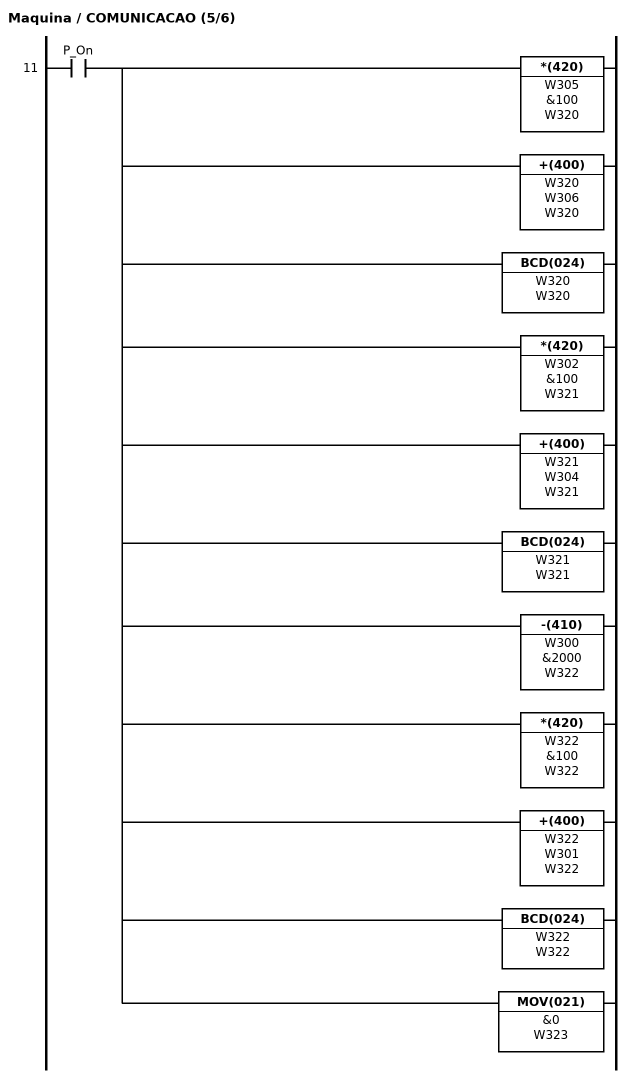
; [picture p24: Maquina / COMUNICACAO, rungs 11-11]
; rung 11
LD P_On
*(420) W305 &100 W320
+(400) W320 W306 W320
BCD(024) W320 W320
*(420) W302 &100 W321
+(400) W321 W304 W321
BCD(024) W321 W321
-(410) W300 &2000 W322
*(420) W322 &100 W322
+(400) W322 W301 W322
BCD(024) W322 W322
MOV(021) &0 W323

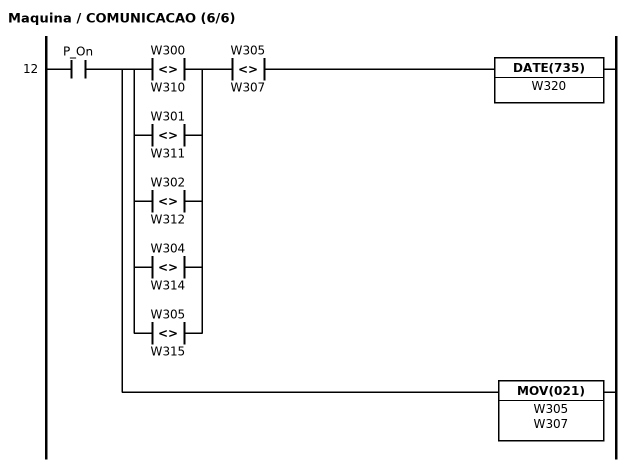
; rung 12
LD P_On
OUT TR0
LD<>(305) W300 W310
OR<>(305) W301 W311
OR<>(305) W302 W312
OR<>(305) W304 W314
OR<>(305) W305 W315
ANDLD
AND<>(305) W305 W307
DATE(735) W320
LD TR0
MOV(021) W305 W307

### Section TASK_CONTROL

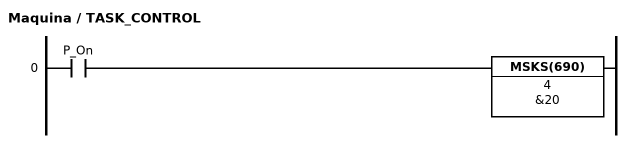
; rung 0
LD P_On
MSKS(690) 4 &20

### Section END
; rung 0
END(001)

## Program Inicializa_strings (cyclic task 127)
Local symbols
ano H130 STRING[2]
data_hora A351 WORD[3]
dia H126 STRING[2]
hora H124 STRING[2]
m_dlog_event_file_name W125 STRING[8]  ; Nome do ficheiro de datalogger
m_dlog_hum_file_name W135 STRING[8]  ; Nome do ficheiro de datalogger
m_dlog_maq_file_name W120 STRING[8]  ; Nome do ficheiro de datalogger
m_dlog_maq_name W110 STRING[10]  ; Nome da maquina
m_dlog_temp_file_name W130 STRING[8]  ; Nome do ficheiro de datalogger
mes H128 STRING[2]
minutos H122 STRING[2]
segundos H120 STRING[2]
str_data_hora H100 STRING[30]  ; String data/hora para datalogger
(*DATA/HORA PARA DATALOGGER*)
IF P_0_1ms=TRUE THEN
	minutos:=left (word_to_string(data_hora[0]),2);
	segundos:=right (word_to_string(data_hora[0]),2);
	dia:=left (word_to_string(data_hora[1]),2);
	hora:=right (word_to_string(data_hora[1]),2);
	ano:=left (word_to_string(data_hora[2]),2);
	mes:=right (word_to_string(data_hora[2]),2);
ELSE
	str_data_hora:= '20'+ano+'-'+mes+'-'+dia+' '+hora+':'+minutos+':'+segundos;
END_IF;

(*NOMES DOS FICHEIROS*)
(*************************************************************************************)

m_dlog_maq_name:= '6';	

m_dlog_maq_file_name:= '\PROG_6';	
m_dlog_event_file_name:= '\EVEN_6';
m_dlog_temp_file_name:= '\TEMP_6';
m_dlog_hum_file_name:= '\HUMI_6';

## Program CAUDAIS (interrupt task 2)
Local symbols
ft01 D700 STRUCT s_caudal  ; Caudalímetro
ft02 D720 STRUCT s_caudal  ; Caudalímetro
ft03 D740 STRUCT s_caudal  ; Caudalímetro
ft04 D760 STRUCT s_caudal  ; Caudalímetro
ft05 D780 STRUCT s_caudal  ; Caudalímetro
om5_injecta 2.15 BOOL  ; Pistola 5
tti1 1.00 BOOL  ; Caudalimetro 1
tti2 1.01 BOOL  ; Caudalimetro 2
tti3 1.02 BOOL  ; Caudalimetro 3
tti4 1.03 BOOL  ; Caudalimetro 4
tti5 1.04 BOOL  ; Caudalimetro 5

### Section M_CAUDAL

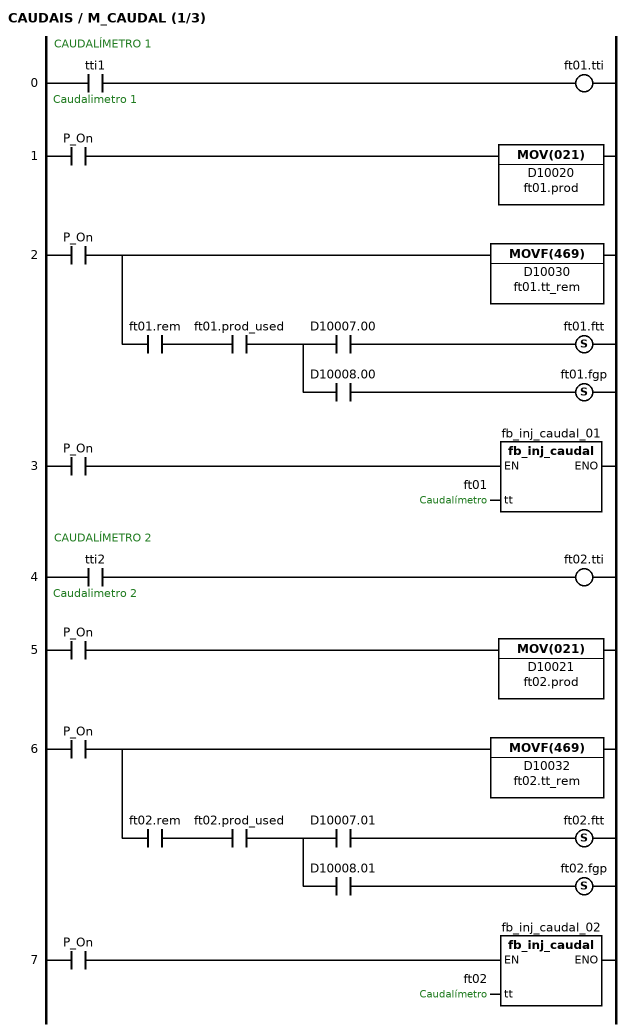
; rung 0: CAUDALÍMETRO 1
!LD tti1  ; Caudalimetro 1
OUT ft01.tti
; rung 1
LD P_On
MOV(021) D10020 ft01.prod
; rung 2
LD P_On
MOVF(469) D10030 ft01.tt_rem
AND ft01.rem
AND ft01.prod_used
OUT TR0
AND D10007.00
SET ft01.ftt
LD TR0
AND D10008.00
SET ft01.fgp
; rung 3
LD P_On
CALL fb_inj_caudal_01 : fb_inj_caudal (tt := ft01)  ; Caudalímetro
; rung 4: CAUDALÍMETRO 2
!LD tti2  ; Caudalimetro 2
OUT ft02.tti
; rung 5
LD P_On
MOV(021) D10021 ft02.prod
; rung 6
LD P_On
MOVF(469) D10032 ft02.tt_rem
AND ft02.rem
AND ft02.prod_used
OUT TR0
AND D10007.01
SET ft02.ftt
LD TR0
AND D10008.01
SET ft02.fgp
; rung 7
LD P_On
CALL fb_inj_caudal_02 : fb_inj_caudal (tt := ft02)  ; Caudalímetro

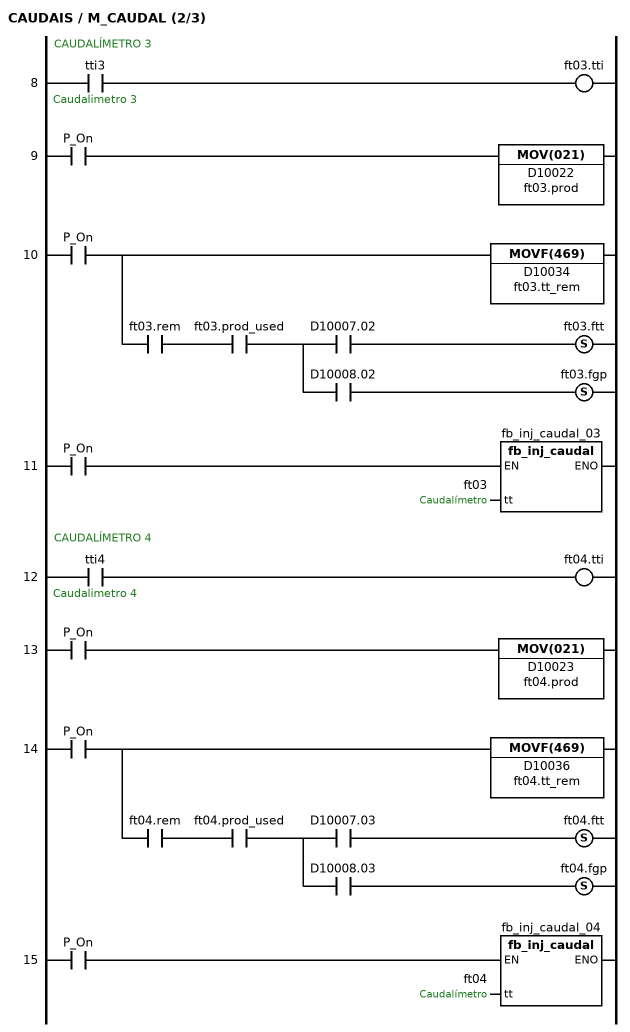
; rung 8: CAUDALÍMETRO 3
!LD tti3  ; Caudalimetro 3
OUT ft03.tti
; rung 9
LD P_On
MOV(021) D10022 ft03.prod
; rung 10
LD P_On
MOVF(469) D10034 ft03.tt_rem
AND ft03.rem
AND ft03.prod_used
OUT TR0
AND D10007.02
SET ft03.ftt
LD TR0
AND D10008.02
SET ft03.fgp
; rung 11
LD P_On
CALL fb_inj_caudal_03 : fb_inj_caudal (tt := ft03)  ; Caudalímetro
; rung 12: CAUDALÍMETRO 4
!LD tti4  ; Caudalimetro 4
OUT ft04.tti
; rung 13
LD P_On
MOV(021) D10023 ft04.prod
; rung 14
LD P_On
MOVF(469) D10036 ft04.tt_rem
AND ft04.rem
AND ft04.prod_used
OUT TR0
AND D10007.03
SET ft04.ftt
LD TR0
AND D10008.03
SET ft04.fgp
; rung 15
LD P_On
CALL fb_inj_caudal_04 : fb_inj_caudal (tt := ft04)  ; Caudalímetro

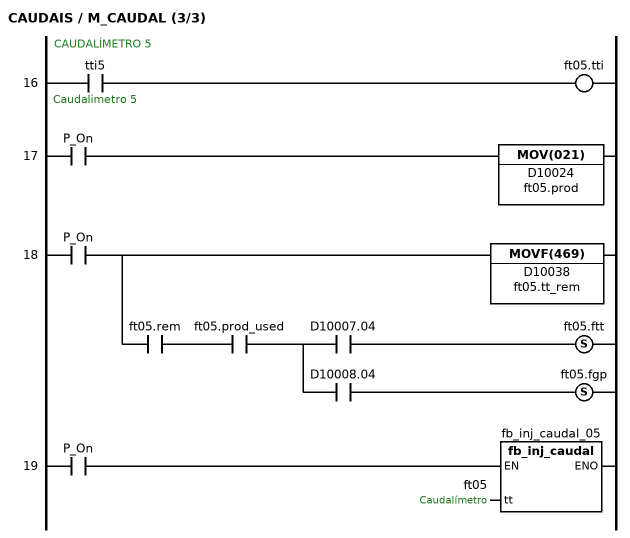
; rung 16: CAUDALÍMETRO 5
!LD tti5  ; Caudalimetro 5
OUT ft05.tti
; rung 17
LD P_On
MOV(021) D10024 ft05.prod
; rung 18
LD P_On
MOVF(469) D10038 ft05.tt_rem
AND ft05.rem
AND ft05.prod_used
OUT TR0
AND D10007.04
SET ft05.ftt
LD TR0
AND D10008.04
SET ft05.fgp
; rung 19
LD P_On
CALL fb_inj_caudal_05 : fb_inj_caudal (tt := ft05)  ; Caudalímetro

### Section END
; rung 0
END(001)

## Function block ExeTimeCalc
VAR_INPUT
  Enable : BOOL;
END_VAR
VAR_OUTPUT
  TotalTime : INT;
  CDT : INT;
END_VAR
VAR_IN_OUT
  prg : s_of_prg;
END_VAR
VAR
  itr : INT;
  ElapsedTime : INT;
  Stp : ARRAY[0..11] OF s_of_pss;
END_VAR
TotalTime:= 0;
ElapsedTime:= 0;

Stp[0].p1:= prg.pss[0].p1; Stp[0].tt:= prg.pss[0].tt; Stp[0].uni:= prg.pss[0].uni;
Stp[1].p1:= prg.pss[1].p1; Stp[1].tt:= prg.pss[1].tt; Stp[1].uni:= prg.pss[1].uni;
Stp[2].p1:= prg.pss[2].p1; Stp[2].tt:= prg.pss[2].tt;Stp[2].uni:= prg.pss[2].uni;
Stp[3].p1:= prg.pss[3].p1; Stp[3].tt:= prg.pss[3].tt; Stp[3].uni:= prg.pss[3].uni;
Stp[4].p1:= prg.pss[4].p1; Stp[4].tt:= prg.pss[4].tt; Stp[4].uni:= prg.pss[4].uni;
Stp[5].p1:= prg.pss[5].p1; Stp[5].tt:= prg.pss[5].tt; Stp[5].uni:= prg.pss[5].uni;
Stp[6].p1:= prg.pss[6].p1; Stp[6].tt:= prg.pss[6].tt; Stp[6].uni:= prg.pss[6].uni;
Stp[7].p1:= prg.pss[7].p1; Stp[7].tt:= prg.pss[7].tt; Stp[7].uni:= prg.pss[7].uni;
Stp[8].p1:= prg.pss[8].p1; Stp[8].tt:= prg.pss[8].tt; Stp[8].uni:= prg.pss[8].uni;
Stp[9].p1:= prg.pss[9].p1; Stp[9].tt:= prg.pss[9].tt; Stp[9].uni:= prg.pss[9].uni;
Stp[10].p1:= prg.pss[10].p1; Stp[10].tt:= prg.pss[10].tt; Stp[10].uni:= prg.pss[10].uni;
Stp[11].p1:= prg.pss[11].p1; Stp[11].tt:= prg.pss[11].tt; Stp[11].uni:= prg.pss[11].uni;

IF Enable THEN
	FOR itr:=0 TO 11 DO
		IF Stp[ itr ].uni=12 THEN
			TotalTime:=TotalTime+ Stp[ itr ].p1;
			ElapsedTime:= ElapsedTime+REAL_TO_INT(Stp[ itr ].tt);
		END_IF;
	END_FOR;
END_IF;
	
CDT := TotalTime - ElapsedTime;

## Function block fb_CopySteps
VAR_INPUT
  Rcp_Ok : BOOL;
END_VAR
VAR_IN_OUT
  Recipe : s_of;
  Steps : ARRAY[0..11] OF s_Steps;
END_VAR
(*Programa*)
Recipe.prg.pss[0].f:=Steps[0].f;
Recipe.prg.pss[0].p1:=Steps[0].p1;
Recipe.prg.pss[0].p2:=Steps[0].p2;
Recipe.prg.pss[0].uni:=0;
Recipe.prg.pss[0].uni:=12;
CASE Recipe.prg.pss[0].f OF
	40:Recipe.prg.pss[0].uni:=9;
END_CASE;

Recipe.prg.pss[1].f:=Steps[1].f;
Recipe.prg.pss[1].p1:=Steps[1].p1;
Recipe.prg.pss[1].p2:=Steps[1].p2;
Recipe.prg.pss[1].uni:=0;
Recipe.prg.pss[1].uni:=12;
CASE Recipe.prg.pss[1].f OF
	40:Recipe.prg.pss[1].uni:=9;
END_CASE;

Recipe.prg.pss[2].f:=Steps[2].f;
Recipe.prg.pss[2].p1:=Steps[2].p1;
Recipe.prg.pss[2].p2:=Steps[2].p2;
Recipe.prg.pss[2].uni:=0;
Recipe.prg.pss[2].uni:=12;
CASE Recipe.prg.pss[2].f OF
	40:Recipe.prg.pss[2].uni:=9;
END_CASE;

Recipe.prg.pss[3].f:=Steps[3].f;
Recipe.prg.pss[3].p1:=Steps[3].p1;
Recipe.prg.pss[3].p2:=Steps[3].p2;
Recipe.prg.pss[3].uni:=0;
Recipe.prg.pss[3].uni:=12;
CASE Recipe.prg.pss[3].f OF
	40:Recipe.prg.pss[3].uni:=9;
END_CASE;

Recipe.prg.pss[4].f:=Steps[4].f;
Recipe.prg.pss[4].p1:=Steps[4].p1;
Recipe.prg.pss[4].p2:=Steps[4].p2;
Recipe.prg.pss[4].uni:=0;
Recipe.prg.pss[4].uni:=12;
CASE Recipe.prg.pss[4].f OF
	40:Recipe.prg.pss[4].uni:=9;
END_CASE;

Recipe.prg.pss[5].f:=Steps[5].f;
Recipe.prg.pss[5].p1:=Steps[5].p1;
Recipe.prg.pss[5].p2:=Steps[5].p2;
Recipe.prg.pss[5].uni:=0;
Recipe.prg.pss[5].uni:=12;
CASE Recipe.prg.pss[5].f OF
	40:Recipe.prg.pss[5].uni:=9;
END_CASE;

Recipe.prg.pss[6].f:=Steps[6].f;
Recipe.prg.pss[6].p1:=Steps[6].p1;
Recipe.prg.pss[6].p2:=Steps[6].p2;
Recipe.prg.pss[6].uni:=0;
Recipe.prg.pss[6].uni:=12;
CASE Recipe.prg.pss[6].f OF
	40:Recipe.prg.pss[6].uni:=9;
END_CASE;

Recipe.prg.pss[7].f:=Steps[7].f;
Recipe.prg.pss[7].p1:=Steps[7].p1;
Recipe.prg.pss[7].p2:=Steps[7].p2;
Recipe.prg.pss[7].uni:=0;
Recipe.prg.pss[7].uni:=12;
CASE Recipe.prg.pss[7].f OF
	40:Recipe.prg.pss[7].uni:=9;
END_CASE;

Recipe.prg.pss[8].f:=Steps[8].f;
Recipe.prg.pss[8].p1:=Steps[8].p1;
Recipe.prg.pss[8].p2:=Steps[8].p2;
Recipe.prg.pss[8].uni:=0;
Recipe.prg.pss[8].uni:=12;
CASE Recipe.prg.pss[8].f OF
	40:Recipe.prg.pss[8].uni:=9;
END_CASE;

Recipe.prg.pss[9].f:=Steps[9].f;
Recipe.prg.pss[9].p1:=Steps[9].p1;
Recipe.prg.pss[9].p2:=Steps[9].p2;
Recipe.prg.pss[9].uni:=0;
Recipe.prg.pss[9].uni:=12;
CASE Recipe.prg.pss[9].f OF
	40:Recipe.prg.pss[9].uni:=9;
END_CASE;

Recipe.prg.pss[10].f:=Steps[9].f;
Recipe.prg.pss[10].p1:=Steps[9].p1;
Recipe.prg.pss[10].p2:=Steps[9].p2;
Recipe.prg.pss[10].uni:=0;
Recipe.prg.pss[10].uni:=12;
CASE Recipe.prg.pss[10].f OF
	40:Recipe.prg.pss[10].uni:=9;
END_CASE;

Recipe.prg.pss[11].f:=Steps[9].f;
Recipe.prg.pss[11].p1:=Steps[9].p1;
Recipe.prg.pss[11].p2:=Steps[9].p2;
Recipe.prg.pss[11].uni:=0;
Recipe.prg.pss[11].uni:=12;
CASE Recipe.prg.pss[11].f OF
	40:Recipe.prg.pss[11].uni:=9;
END_CASE;

Recipe.dados:= Rcp_Ok;

## Function block fb_f_aquece
; FUNÇÃO AQUECIMENTO USANDO TC104 - Faz a função de aquecimento usando uma carta TC104 com PID
VAR_IN_OUT
  maq : s_maquina;  (* Dados da maquina *)
  aquece : s_f_aquece;  (* Dados da função de aquecimento *)
  aspira : s_f_aspira;  (* Dados da função de aspiração *)
END_VAR
VAR
  tm01 : TIMER;
  sp_hh : REAL;  (* Valor superior do setpoint *)
  sp_ll : REAL;  (* Valor inferior do setpoint *)
  p1 : REAL;  (* Parametro 1 da função em REAL *)
  sp_ft : UDINT;
  tm02 : TIMER;
  tm03 : TIMER;
  tm04 : TIMER;
  p1_end : REAL;  (* Valor apartir do qual deixa de aquecer. *)
END_VAR

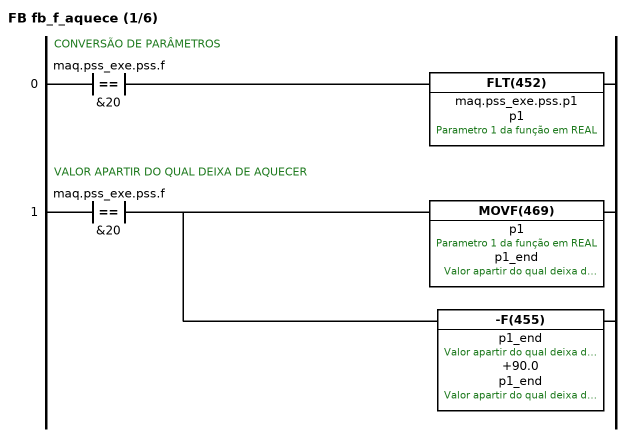
; rung 0: CONVERSÃO DE PARÂMETROS
LD=(300) maq.pss_exe.pss.f &20
FLT(452) maq.pss_exe.pss.p1 p1  ; Parametro 1 da função em REAL
; rung 1: VALOR APARTIR DO QUAL DEIXA DE AQUECER
LD=(300) maq.pss_exe.pss.f &20
MOVF(469) p1 p1_end  ; Parametro 1 da função em REAL, Valor apartir do qual deixa de aquecer.
-F(455) p1_end +90.0 p1_end  ; Valor apartir do qual deixa de aquecer.

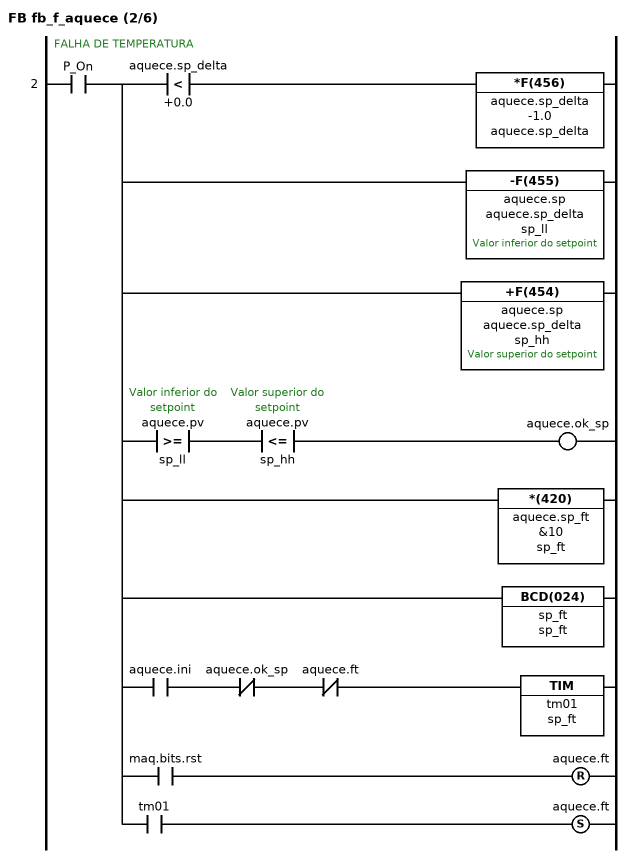
; rung 2: FALHA DE TEMPERATURA
LD P_On
OUT TR0
AND<F(331) aquece.sp_delta +0.0
*F(456) aquece.sp_delta -1.0 aquece.sp_delta
LD TR0
-F(455) aquece.sp aquece.sp_delta sp_ll  ; Valor inferior do setpoint
+F(454) aquece.sp aquece.sp_delta sp_hh  ; Valor superior do setpoint
AND>=F(334) aquece.pv sp_ll  ; Valor inferior do setpoint
AND<=F(332) aquece.pv sp_hh  ; Valor superior do setpoint
OUT aquece.ok_sp
LD TR0
*(420) aquece.sp_ft &10 sp_ft
BCD(024) sp_ft sp_ft
AND aquece.ini
ANDNOT aquece.ok_sp
ANDNOT aquece.ft
TIM tm01 sp_ft
LD TR0
AND maq.bits.rst
RSET aquece.ft
LD TR0
AND tm01
SET aquece.ft

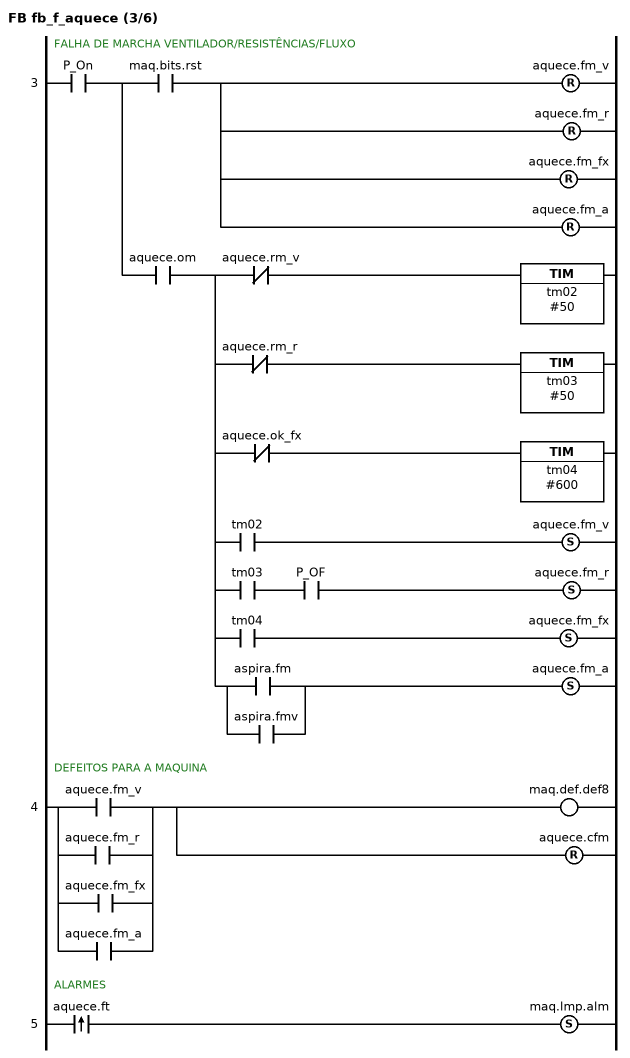
; rung 3: FALHA DE MARCHA VENTILADOR/RESISTÊNCIAS/FLUXO
LD P_On
OUT TR0
AND maq.bits.rst
RSET aquece.fm_v
RSET aquece.fm_r
RSET aquece.fm_fx
RSET aquece.fm_a
LD TR0
AND aquece.om
OUT TR1
ANDNOT aquece.rm_v
TIM tm02 #50
LD TR1
ANDNOT aquece.rm_r
TIM tm03 #50
LD TR1
ANDNOT aquece.ok_fx
TIM tm04 #600
LD TR1
AND tm02
SET aquece.fm_v
LD TR1
AND tm03
AND P_OF
SET aquece.fm_r
LD TR1
AND tm04
SET aquece.fm_fx
LD TR1
LD aspira.fm
OR aspira.fmv
ANDLD
SET aquece.fm_a
; rung 4: DEFEITOS PARA A MAQUINA
LD aquece.fm_v
OR aquece.fm_r
OR aquece.fm_fx
OR aquece.fm_a
OUT maq.def.def8
RSET aquece.cfm
; rung 5: ALARMES
@LD aquece.ft
SET maq.lmp.alm

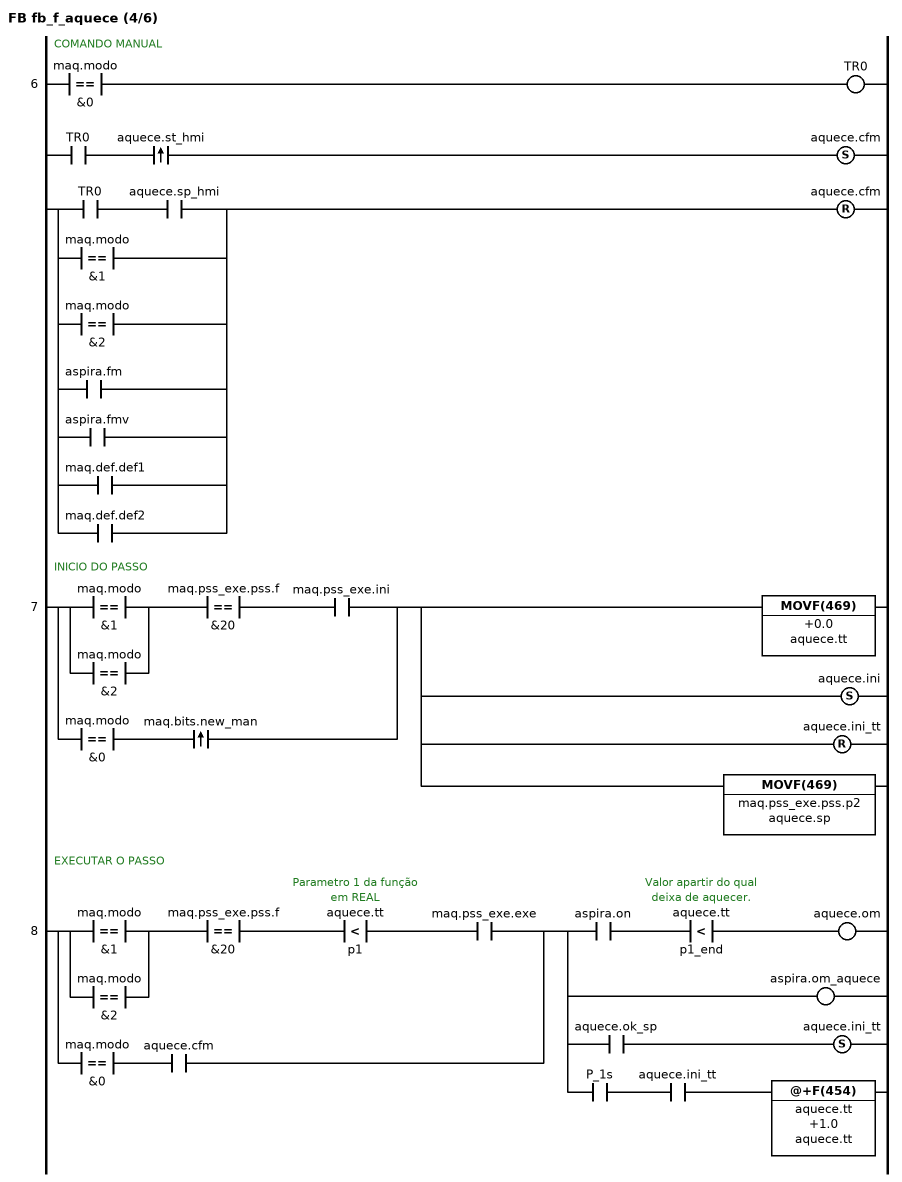
; rung 6: COMANDO MANUAL
LD=(300) maq.modo &0
OUT TR0
LD TR0
@AND aquece.st_hmi
SET aquece.cfm
LD TR0
AND aquece.sp_hmi
OR=(300) maq.modo &1
OR=(300) maq.modo &2
OR aspira.fm
OR aspira.fmv
OR maq.def.def1
OR maq.def.def2
RSET aquece.cfm
; rung 7: INICIO DO PASSO
LD=(300) maq.modo &1
OR=(300) maq.modo &2
AND=(300) maq.pss_exe.pss.f &20
AND maq.pss_exe.ini
LD=(300) maq.modo &0
@AND maq.bits.new_man
ORLD
MOVF(469) +0.0 aquece.tt
SET aquece.ini
RSET aquece.ini_tt
MOVF(469) maq.pss_exe.pss.p2 aquece.sp
; rung 8: EXECUTAR O PASSO
LD=(300) maq.modo &1
OR=(300) maq.modo &2
AND=(300) maq.pss_exe.pss.f &20
AND<F(331) aquece.tt p1  ; Parametro 1 da função em REAL
AND maq.pss_exe.exe
LD=(300) maq.modo &0
AND aquece.cfm
ORLD
OUT TR0
AND aspira.on
AND<F(331) aquece.tt p1_end  ; Valor apartir do qual deixa de aquecer.
OUT aquece.om
LD TR0
OUT aspira.om_aquece
AND aquece.ok_sp
SET aquece.ini_tt
LD TR0
AND P_1s
AND aquece.ini_tt
@+F(454) aquece.tt +1.0 aquece.tt

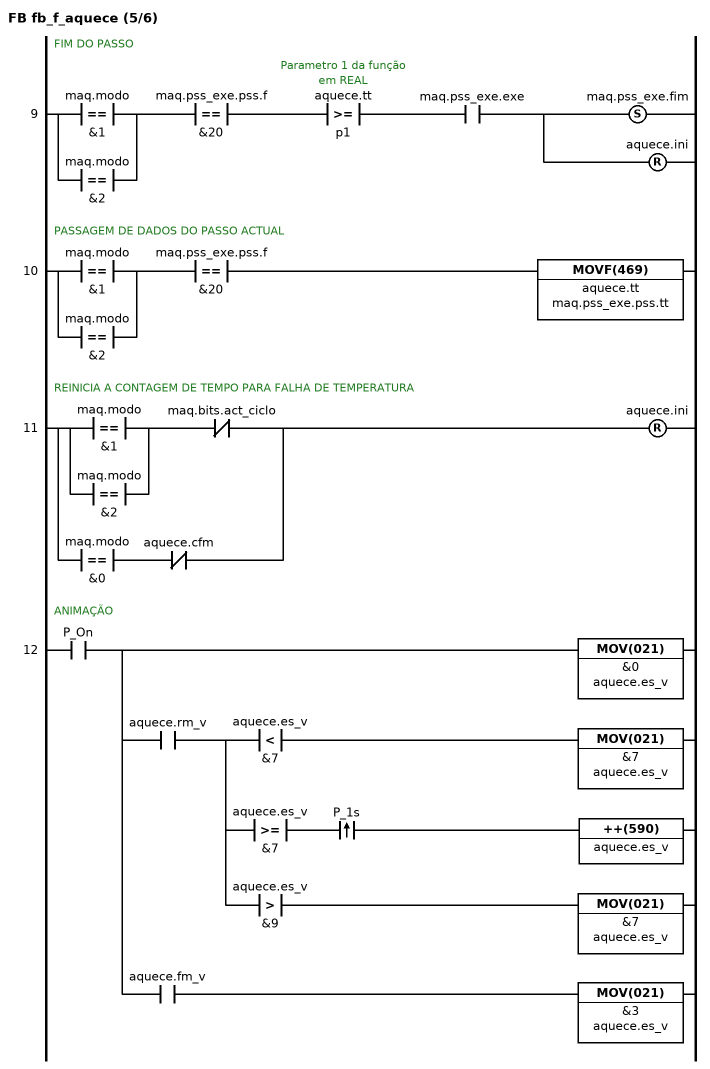
; rung 9: FIM DO PASSO
LD=(300) maq.modo &1
OR=(300) maq.modo &2
AND=(300) maq.pss_exe.pss.f &20
AND>=F(334) aquece.tt p1  ; Parametro 1 da função em REAL
AND maq.pss_exe.exe
SET maq.pss_exe.fim
RSET aquece.ini
; rung 10: PASSAGEM DE DADOS DO PASSO ACTUAL
LD=(300) maq.modo &1
OR=(300) maq.modo &2
AND=(300) maq.pss_exe.pss.f &20
MOVF(469) aquece.tt maq.pss_exe.pss.tt
; rung 11: REINICIA A CONTAGEM DE TEMPO PARA FALHA DE TEMPERATURA
LD=(300) maq.modo &1
OR=(300) maq.modo &2
ANDNOT maq.bits.act_ciclo
LD=(300) maq.modo &0
ANDNOT aquece.cfm
ORLD
RSET aquece.ini
; rung 12: ANIMAÇÃO
LD P_On
OUT TR0
MOV(021) &0 aquece.es_v
AND aquece.rm_v
OUT TR1
AND<(310) aquece.es_v &7
MOV(021) &7 aquece.es_v
LD TR1
AND>=(325) aquece.es_v &7
@AND P_1s
++(590) aquece.es_v
LD TR1
AND>(320) aquece.es_v &9
MOV(021) &7 aquece.es_v
LD TR0
AND aquece.fm_v
MOV(021) &3 aquece.es_v

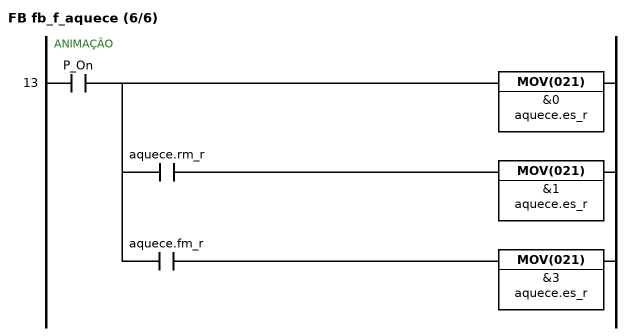
; rung 13: ANIMAÇÃO
LD P_On
OUT TR0
MOV(021) &0 aquece.es_r
AND aquece.rm_r
MOV(021) &1 aquece.es_r
LD TR0
AND aquece.fm_r
MOV(021) &3 aquece.es_r

## Function block fb_f_aspira
; FUNÇÃO ASPIRAÇÃO - Faz a função de aspiração. Controlo de inputs/outputs
VAR_IN_OUT
  maq : s_maquina;  (* Dados da maquina *)
  aspira : s_f_aspira;  (* Dados da função de aspiração *)
END_VAR
VAR
  tm01 : TIMER;
  tm02 : TIMER;
  p1 : REAL;  (* Parametro 1 da função em REAL *)
  tm03 : TIMER;
END_VAR

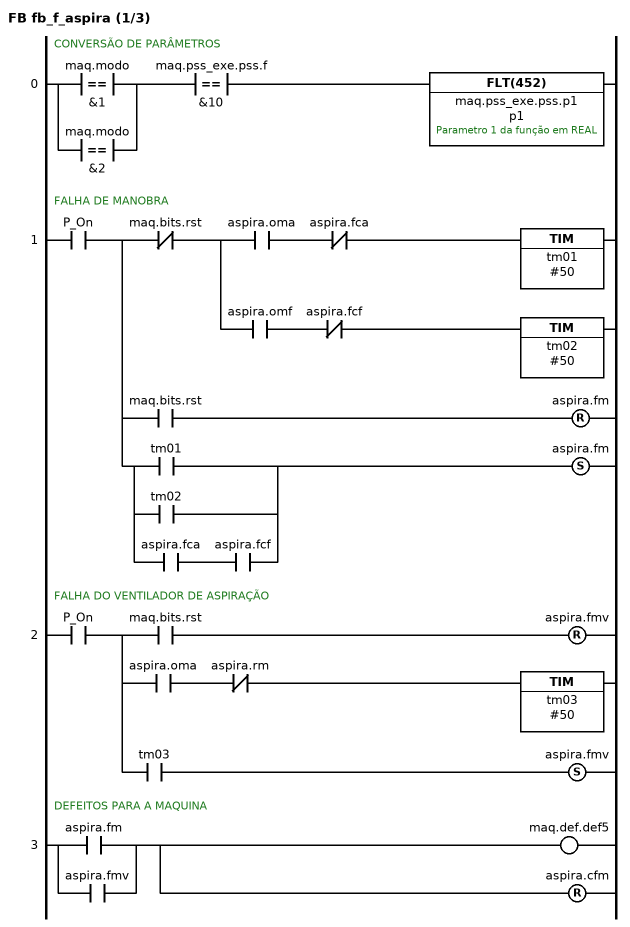
; rung 0: CONVERSÃO DE PARÂMETROS
LD=(300) maq.modo &1
OR=(300) maq.modo &2
AND=(300) maq.pss_exe.pss.f &10
FLT(452) maq.pss_exe.pss.p1 p1  ; Parametro 1 da função em REAL
; rung 1: FALHA DE MANOBRA
LD P_On
OUT TR0
ANDNOT maq.bits.rst
OUT TR1
AND aspira.oma
ANDNOT aspira.fca
TIM tm01 #50
LD TR1
AND aspira.omf
ANDNOT aspira.fcf
TIM tm02 #50
LD TR0
AND maq.bits.rst
RSET aspira.fm
LD TR0
LD tm01
OR tm02
LD aspira.fca
AND aspira.fcf
ORLD
ANDLD
SET aspira.fm
; rung 2: FALHA DO VENTILADOR DE ASPIRAÇÃO
LD P_On
OUT TR0
AND maq.bits.rst
RSET aspira.fmv
LD TR0
AND aspira.oma
ANDNOT aspira.rm
TIM tm03 #50
LD TR0
AND tm03
SET aspira.fmv
; rung 3: DEFEITOS PARA A MAQUINA
LD aspira.fm
OR aspira.fmv
OUT maq.def.def5
RSET aspira.cfm

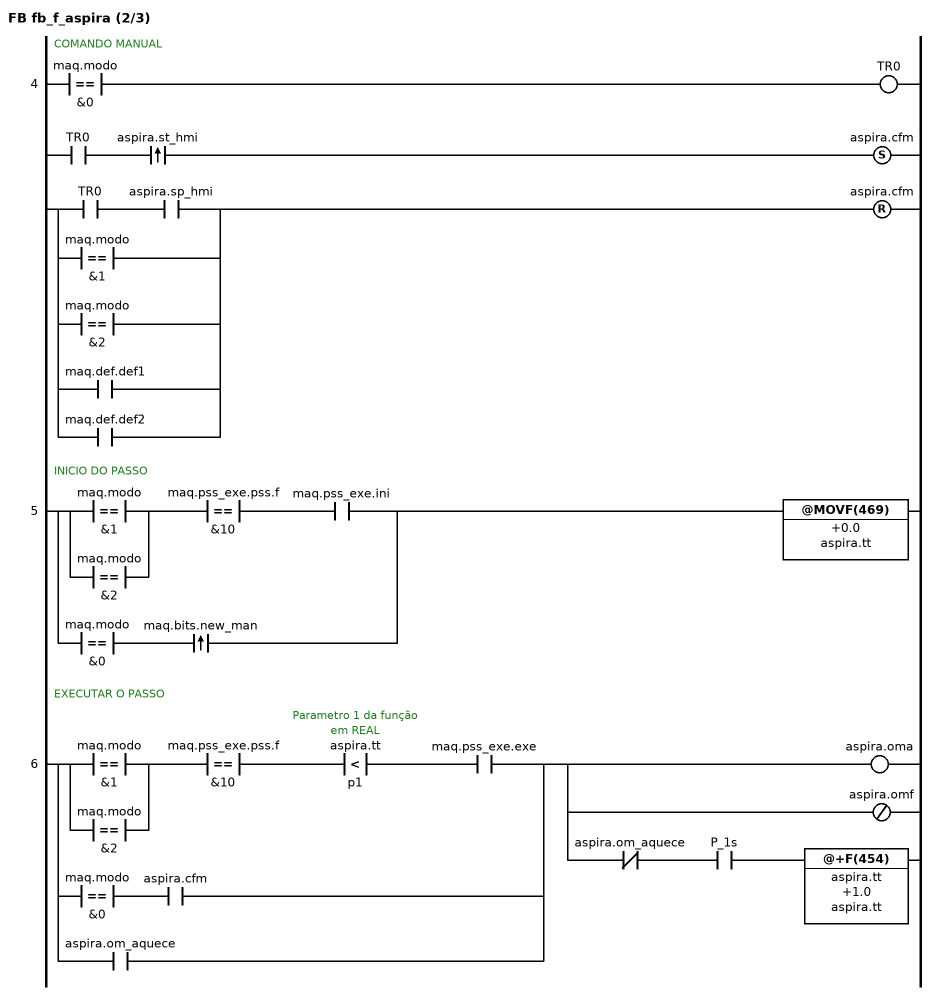
; rung 4: COMANDO MANUAL
LD=(300) maq.modo &0
OUT TR0
LD TR0
@AND aspira.st_hmi
SET aspira.cfm
LD TR0
AND aspira.sp_hmi
OR=(300) maq.modo &1
OR=(300) maq.modo &2
OR maq.def.def1
OR maq.def.def2
RSET aspira.cfm
; rung 5: INICIO DO PASSO
LD=(300) maq.modo &1
OR=(300) maq.modo &2
AND=(300) maq.pss_exe.pss.f &10
AND maq.pss_exe.ini
LD=(300) maq.modo &0
@AND maq.bits.new_man
ORLD
@MOVF(469) +0.0 aspira.tt
; rung 6: EXECUTAR O PASSO
LD=(300) maq.modo &1
OR=(300) maq.modo &2
AND=(300) maq.pss_exe.pss.f &10
AND<F(331) aspira.tt p1  ; Parametro 1 da função em REAL
AND maq.pss_exe.exe
LD=(300) maq.modo &0
AND aspira.cfm
ORLD
OR aspira.om_aquece
OUT aspira.oma
OUTNOT aspira.omf
ANDNOT aspira.om_aquece
AND P_1s
@+F(454) aspira.tt +1.0 aspira.tt

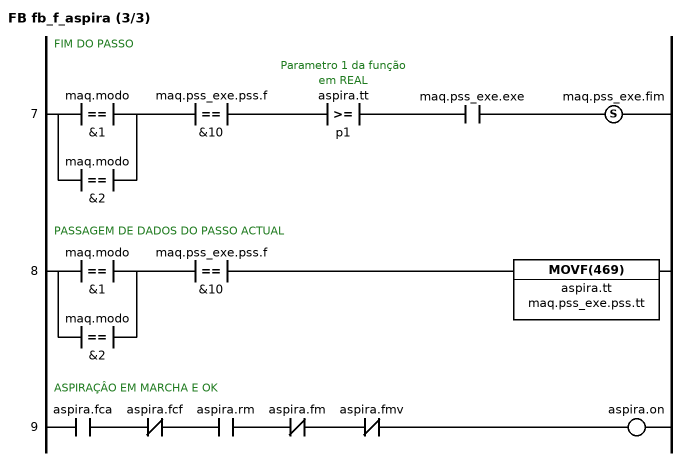
; rung 7: FIM DO PASSO
LD=(300) maq.modo &1
OR=(300) maq.modo &2
AND=(300) maq.pss_exe.pss.f &10
AND>=F(334) aspira.tt p1  ; Parametro 1 da função em REAL
AND maq.pss_exe.exe
SET maq.pss_exe.fim
; rung 8: PASSAGEM DE DADOS DO PASSO ACTUAL
LD=(300) maq.modo &1
OR=(300) maq.modo &2
AND=(300) maq.pss_exe.pss.f &10
MOVF(469) aspira.tt maq.pss_exe.pss.tt
; rung 9: ASPIRAÇÂO EM MARCHA E OK
LD aspira.fca
ANDNOT aspira.fcf
AND aspira.rm
ANDNOT aspira.fm
ANDNOT aspira.fmv
OUT aspira.on

## Function block fb_f_injecta
; FUNÇÃO INJECÇÃO - Faz a função de injecção
VAR_IN_OUT
  maq : s_maquina;  (* Dados da maquina *)
  injecta : s_f_injecta;  (* Dados da função de injecção *)
  caudal : s_caudal;  (* Dados do caudalímetro *)
END_VAR
VAR
  tm01 : TIMER;
END_VAR

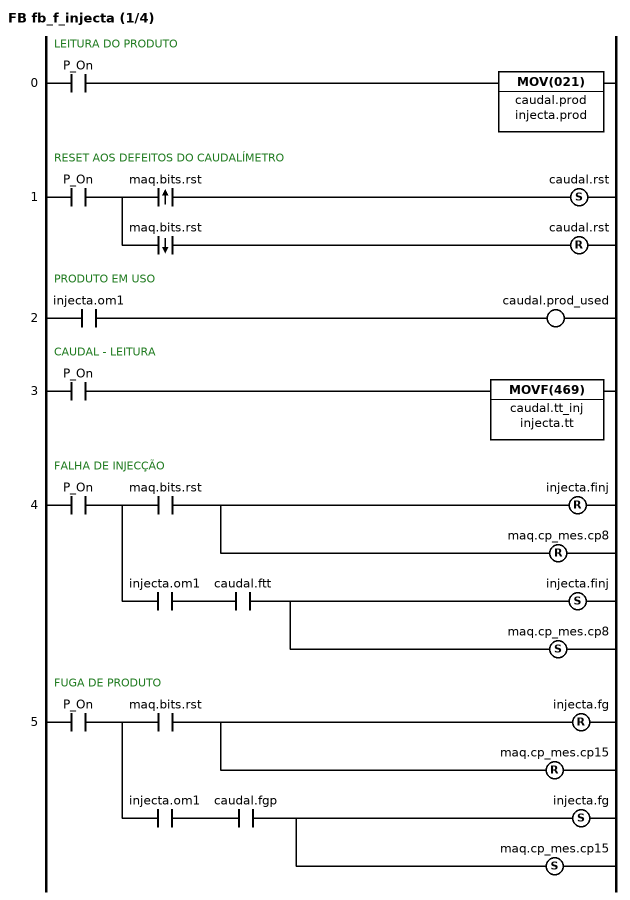
; rung 0: LEITURA DO PRODUTO
LD P_On
MOV(021) caudal.prod injecta.prod
; rung 1: RESET AOS DEFEITOS DO CAUDALÍMETRO
LD P_On
OUT TR0
@AND maq.bits.rst
SET caudal.rst
LD TR0
%AND maq.bits.rst
RSET caudal.rst
; rung 2: PRODUTO EM USO
LD injecta.om1
OUT caudal.prod_used
; rung 3: CAUDAL - LEITURA
LD P_On
MOVF(469) caudal.tt_inj injecta.tt
; rung 4: FALHA DE INJECÇÃO
LD P_On
OUT TR0
AND maq.bits.rst
RSET injecta.finj
RSET maq.cp_mes.cp8
LD TR0
AND injecta.om1
AND caudal.ftt
SET injecta.finj
SET maq.cp_mes.cp8
; rung 5: FUGA DE PRODUTO
LD P_On
OUT TR0
AND maq.bits.rst
RSET injecta.fg
RSET maq.cp_mes.cp15
LD TR0
AND injecta.om1
AND caudal.fgp
SET injecta.fg
SET maq.cp_mes.cp15

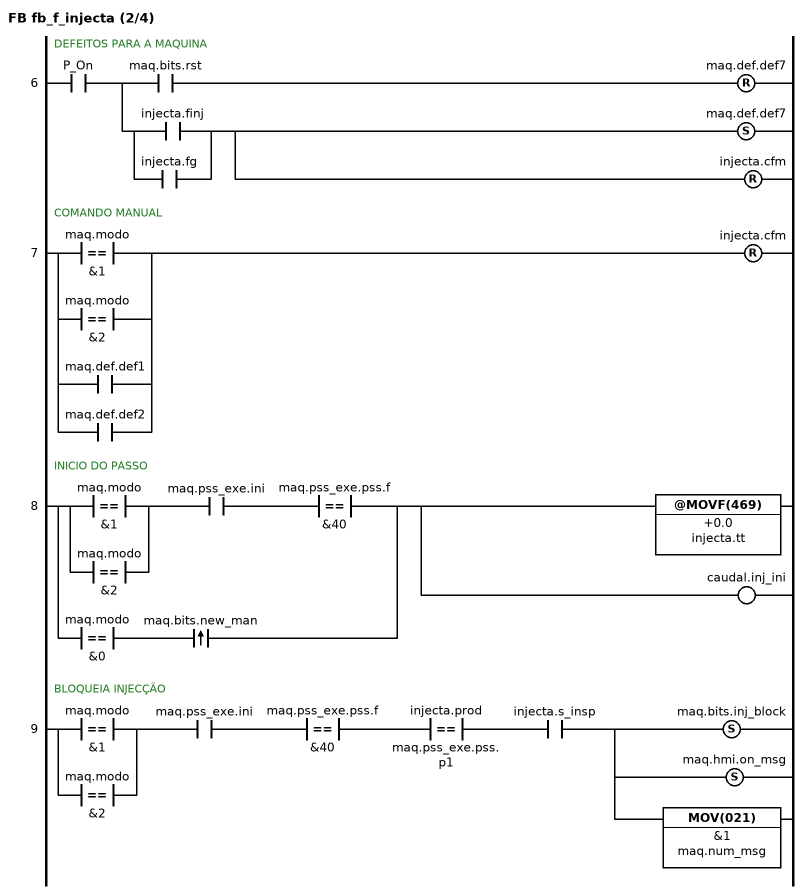
; rung 6: DEFEITOS PARA A MAQUINA
LD P_On
OUT TR0
AND maq.bits.rst
RSET maq.def.def7
LD TR0
LD injecta.finj
OR injecta.fg
ANDLD
SET maq.def.def7
RSET injecta.cfm
; rung 7: COMANDO MANUAL
LD=(300) maq.modo &1
OR=(300) maq.modo &2
OR maq.def.def1
OR maq.def.def2
RSET injecta.cfm
; rung 8: INICIO DO PASSO
LD=(300) maq.modo &1
OR=(300) maq.modo &2
AND maq.pss_exe.ini
AND=(300) maq.pss_exe.pss.f &40
LD=(300) maq.modo &0
@AND maq.bits.new_man
ORLD
@MOVF(469) +0.0 injecta.tt
OUT caudal.inj_ini
; rung 9: BLOQUEIA INJECÇÃO
LD=(300) maq.modo &1
OR=(300) maq.modo &2
AND maq.pss_exe.ini
AND=(300) maq.pss_exe.pss.f &40
AND=(300) injecta.prod maq.pss_exe.pss.p1
AND injecta.s_insp
SET maq.bits.inj_block
SET maq.hmi.on_msg
MOV(021) &1 maq.num_msg

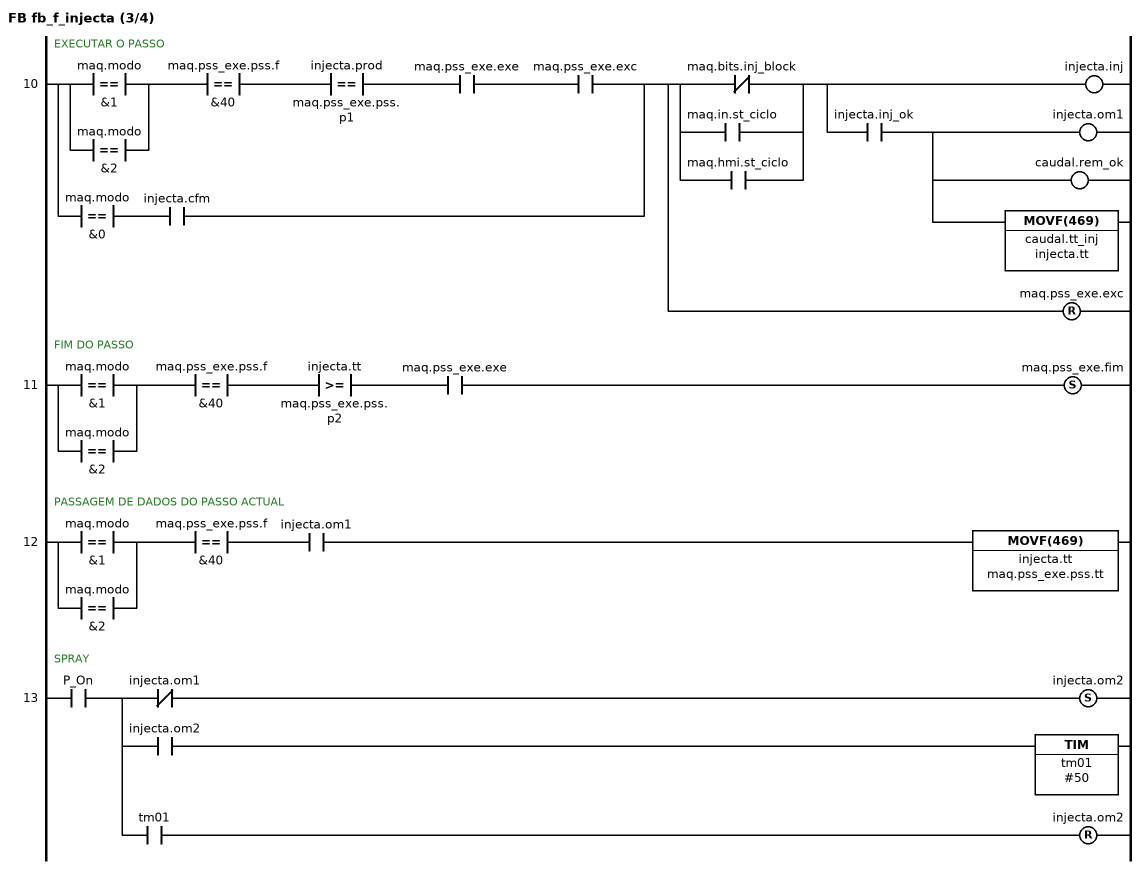
; rung 10: EXECUTAR O PASSO
LD=(300) maq.modo &1
OR=(300) maq.modo &2
AND=(300) maq.pss_exe.pss.f &40
AND=(300) injecta.prod maq.pss_exe.pss.p1
AND maq.pss_exe.exe
AND maq.pss_exe.exc
LD=(300) maq.modo &0
AND injecta.cfm
ORLD
OUT TR0
LDNOT maq.bits.inj_block
OR maq.in.st_ciclo
OR maq.hmi.st_ciclo
ANDLD
OUT injecta.inj
AND injecta.inj_ok
OUT injecta.om1
OUT caudal.rem_ok
MOVF(469) caudal.tt_inj injecta.tt
LD TR0
RSET maq.pss_exe.exc
; rung 11: FIM DO PASSO
LD=(300) maq.modo &1
OR=(300) maq.modo &2
AND=(300) maq.pss_exe.pss.f &40
AND>=F(334) injecta.tt maq.pss_exe.pss.p2
AND maq.pss_exe.exe
SET maq.pss_exe.fim
; rung 12: PASSAGEM DE DADOS DO PASSO ACTUAL
LD=(300) maq.modo &1
OR=(300) maq.modo &2
AND=(300) maq.pss_exe.pss.f &40
AND injecta.om1
MOVF(469) injecta.tt maq.pss_exe.pss.tt
; rung 13: SPRAY
LD P_On
OUT TR0
ANDNOT injecta.om1
SET injecta.om2
LD TR0
AND injecta.om2
TIM tm01 #50
LD TR0
AND tm01
RSET injecta.om2

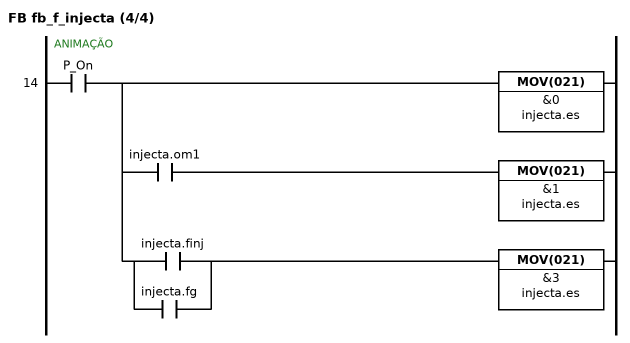
; rung 14: ANIMAÇÃO
LD P_On
OUT TR0
MOV(021) &0 injecta.es
AND injecta.om1
MOV(021) &1 injecta.es
LD TR0
LD injecta.finj
OR injecta.fg
ANDLD
MOV(021) &3 injecta.es

## Function block fb_f_injecta_man
; FUNÇÃO INJECÇÃO MANUAL - Faz a função de injecção manual (chamar após injecção auto)
VAR_IN_OUT
  maq : s_maquina;  (* Dados da maquina *)
END_VAR

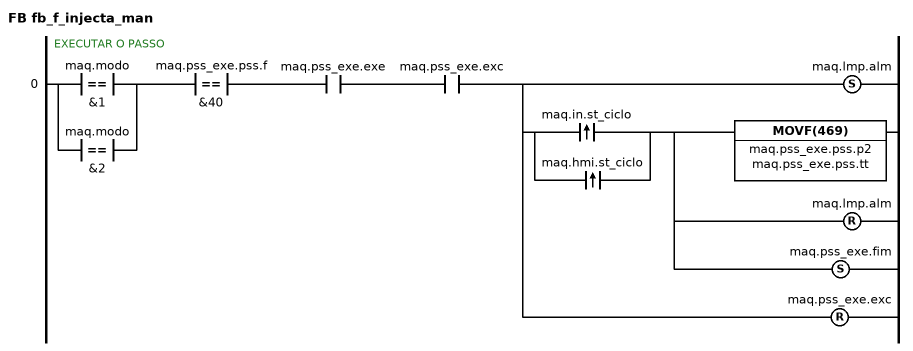
; rung 0: EXECUTAR O PASSO
LD=(300) maq.modo &1
OR=(300) maq.modo &2
AND=(300) maq.pss_exe.pss.f &40
AND maq.pss_exe.exe
AND maq.pss_exe.exc
OUT TR0
SET maq.lmp.alm
@LD maq.in.st_ciclo
@OR maq.hmi.st_ciclo
ANDLD
MOVF(469) maq.pss_exe.pss.p2 maq.pss_exe.pss.tt
RSET maq.lmp.alm
SET maq.pss_exe.fim
LD TR0
RSET maq.pss_exe.exc

## Function block fb_f_trata
; FUNÇÃO TRATAMENTO - Faz a função de tratamento. Controlo de inputs/outputs
VAR_IN_OUT
  maq : s_maquina;  (* Dados da maquina *)
  trata : s_f_trata;  (* Dados da função de tratamento *)
END_VAR
VAR
  tm01 : TIMER;
  tm02 : TIMER;
  p1 : REAL;  (* Parametro 1 da função em REAL *)
  tm03 : TIMER;
END_VAR

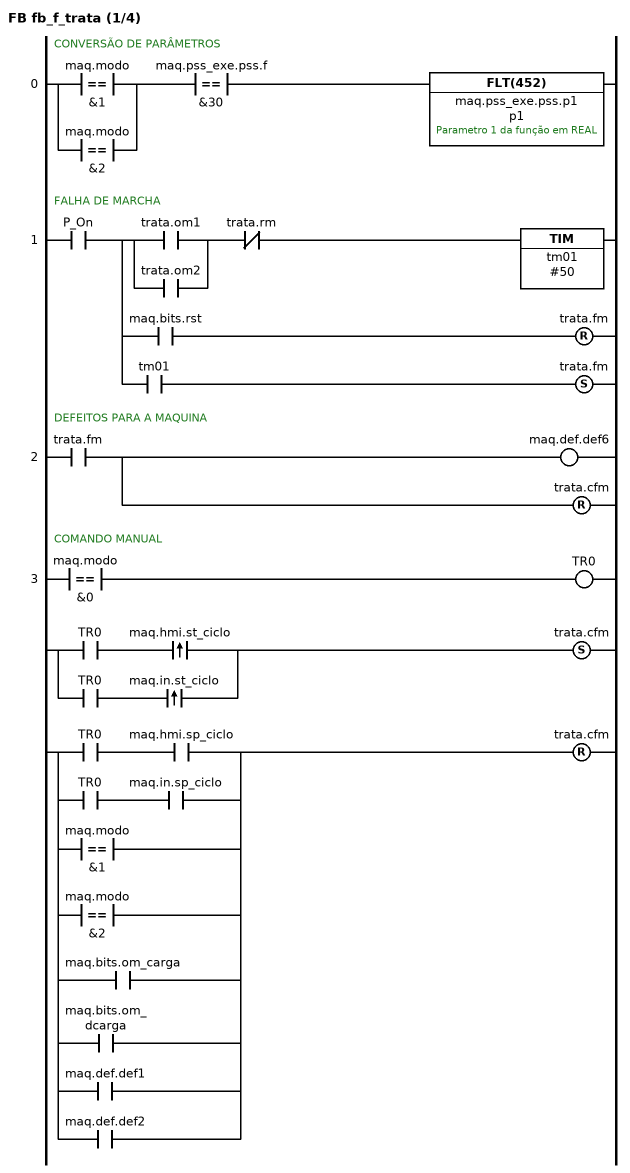
; rung 0: CONVERSÃO DE PARÂMETROS
LD=(300) maq.modo &1
OR=(300) maq.modo &2
AND=(300) maq.pss_exe.pss.f &30
FLT(452) maq.pss_exe.pss.p1 p1  ; Parametro 1 da função em REAL
; rung 1: FALHA DE MARCHA
LD P_On
OUT TR0
LD trata.om1
OR trata.om2
ANDLD
ANDNOT trata.rm
TIM tm01 #50
LD TR0
AND maq.bits.rst
RSET trata.fm
LD TR0
AND tm01
SET trata.fm
; rung 2: DEFEITOS PARA A MAQUINA
LD trata.fm
OUT maq.def.def6
RSET trata.cfm
; rung 3: COMANDO MANUAL
LD=(300) maq.modo &0
OUT TR0
LD TR0
@AND maq.hmi.st_ciclo
LD TR0
@AND maq.in.st_ciclo
ORLD
SET trata.cfm
LD TR0
AND maq.hmi.sp_ciclo
LD TR0
AND maq.in.sp_ciclo
ORLD
OR=(300) maq.modo &1
OR=(300) maq.modo &2
OR maq.bits.om_carga
OR maq.bits.om_dcarga
OR maq.def.def1
OR maq.def.def2
RSET trata.cfm

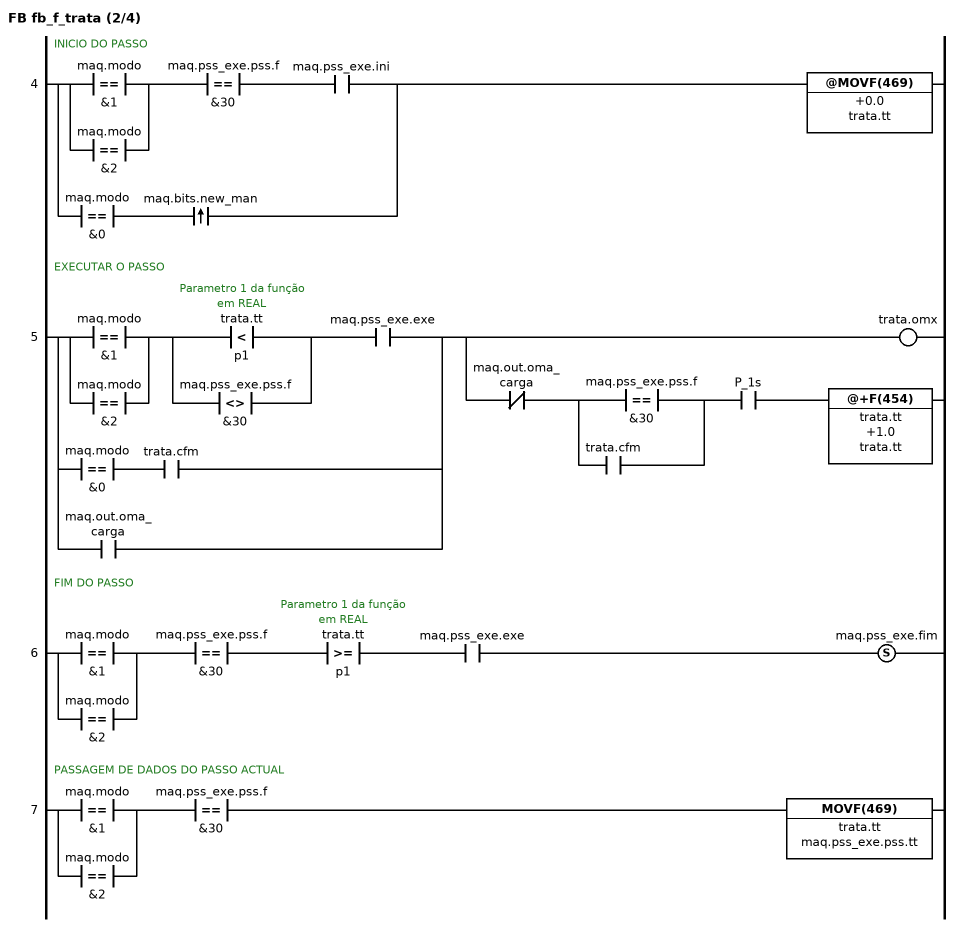
; rung 4: INICIO DO PASSO
LD=(300) maq.modo &1
OR=(300) maq.modo &2
AND=(300) maq.pss_exe.pss.f &30
AND maq.pss_exe.ini
LD=(300) maq.modo &0
@AND maq.bits.new_man
ORLD
@MOVF(469) +0.0 trata.tt
; rung 5: EXECUTAR O PASSO
LD=(300) maq.modo &1
OR=(300) maq.modo &2
LD<F(331) trata.tt p1  ; Parametro 1 da função em REAL
OR<>(305) maq.pss_exe.pss.f &30
ANDLD
AND maq.pss_exe.exe
LD=(300) maq.modo &0
AND trata.cfm
ORLD
OR maq.out.oma_carga
OUT trata.omx
ANDNOT maq.out.oma_carga
LD=(300) maq.pss_exe.pss.f &30
OR trata.cfm
ANDLD
AND P_1s
@+F(454) trata.tt +1.0 trata.tt
; rung 6: FIM DO PASSO
LD=(300) maq.modo &1
OR=(300) maq.modo &2
AND=(300) maq.pss_exe.pss.f &30
AND>=F(334) trata.tt p1  ; Parametro 1 da função em REAL
AND maq.pss_exe.exe
SET maq.pss_exe.fim
; rung 7: PASSAGEM DE DADOS DO PASSO ACTUAL
LD=(300) maq.modo &1
OR=(300) maq.modo &2
AND=(300) maq.pss_exe.pss.f &30
MOVF(469) trata.tt maq.pss_exe.pss.tt

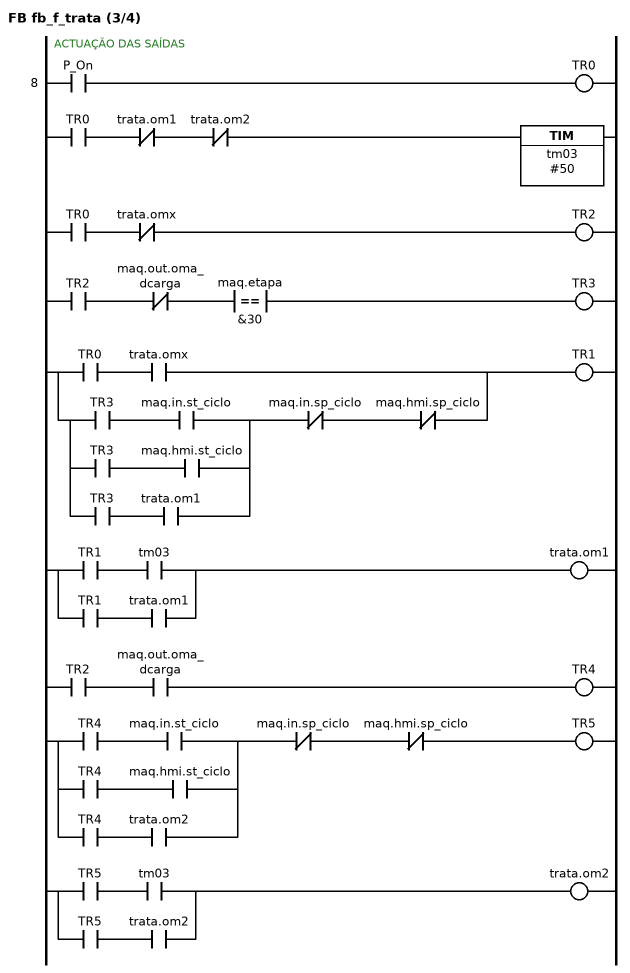
; rung 8: ACTUAÇÃO DAS SAÍDAS
LD P_On
OUT TR0
LD TR0
ANDNOT trata.om1
ANDNOT trata.om2
TIM tm03 #50
LD TR0
ANDNOT trata.omx
OUT TR2
LD TR2
ANDNOT maq.out.oma_dcarga
AND=(300) maq.etapa &30
OUT TR3
LD TR0
AND trata.omx
LD TR3
AND maq.in.st_ciclo
LD TR3
AND maq.hmi.st_ciclo
ORLD
LD TR3
AND trata.om1
ORLD
ANDNOT maq.in.sp_ciclo
ANDNOT maq.hmi.sp_ciclo
ORLD
OUT TR1
LD TR1
AND tm03
LD TR1
AND trata.om1
ORLD
OUT trata.om1
LD TR2
AND maq.out.oma_dcarga
OUT TR4
LD TR4
AND maq.in.st_ciclo
LD TR4
AND maq.hmi.st_ciclo
ORLD
LD TR4
AND trata.om2
ORLD
ANDNOT maq.in.sp_ciclo
ANDNOT maq.hmi.sp_ciclo
OUT TR5
LD TR5
AND tm03
LD TR5
AND trata.om2
ORLD
OUT trata.om2

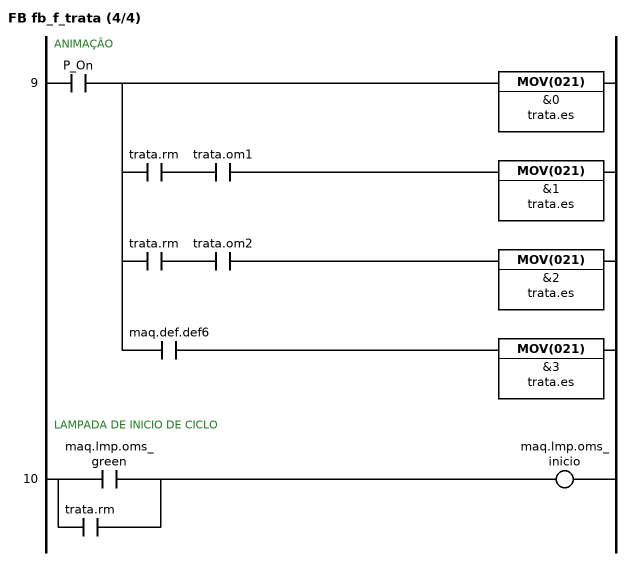
; rung 9: ANIMAÇÃO
LD P_On
OUT TR0
MOV(021) &0 trata.es
AND trata.rm
AND trata.om1
MOV(021) &1 trata.es
LD TR0
AND trata.rm
AND trata.om2
MOV(021) &2 trata.es
LD TR0
AND maq.def.def6
MOV(021) &3 trata.es
; rung 10: LAMPADA DE INICIO DE CICLO
LD maq.lmp.oms_green
OR trata.rm
OUT maq.lmp.oms_inicio

## Function block fb_inj_carro
; FUNÇÃO CARRO DE INJECÇÃO - Controla o funcionamento do carro de injecção, recebendo ordem e enviando permissão às pistolas.
VAR_IN_OUT
  maq : s_maquina;  (* Dados da maquina *)
  carro : s_carro;  (* Dados do carrinho *)
END_VAR
VAR
  cal_fcr : BOOL;  (* Calibração - Fim de curso de recuo atingido *)
  cal_fca : BOOL;  (* Calibração - Fim de curso de avanço atingido *)
  lim_max : BOOL;  (* Limites - Maximo *)
  lim_min : BOOL;  (* Limites - Minimo *)
  om : BOOL;  (* Ordem de marcha *)
  omr : BOOL;  (* Ordem de marcha recuo *)
  tm01 : TIMER;
  tm02 : TIMER;
  tm03 : TIMER;
  r1 : REAL;  (* Auxiliar Real *)
  r2 : REAL;  (* Auxiliar Real *)
END_VAR

